FUNCTION SI : LREAL
VAR_INPUT
	x	: LREAL;
END_VAR
VAR
END_VAR

IF (x > -0.001) AND (x < 0.001) THEN
	SI := 1.0;
ELSE
	SI := SIN(x) / x;
END_IF

END_FUNCTION

(* stored: Version 1.1.0.1, ProductVersion 3.1.4024.11
   POU SI: Id {df8897c1-e126-495b-8643-b65e708f885c}, SpecialFunc None *)
